(* IEC 61131-3 sources: project_Secure_SCADA/rel_v1.2, 1 file *)

(* ---- rel_v1.2.st ---- *)
FUNCTION_BLOCK TP_WITH_RESET
  VAR_INPUT
    IN : BOOL;
    PT : TIME;
    RESET : BOOL;
  END_VAR
  VAR_OUTPUT
    Q : BOOL;
    ET : TIME := T#0s;
  END_VAR
  VAR
    STATE : SINT := 0;
    PREV_IN : BOOL := FALSE;
    CURRENT_TIME : TIME;
    START_TIME : TIME;
  END_VAR

  (* Pragma to set current time *)
  {__SET_VAR(data__->,CURRENT_TIME,,__CURRENT_TIME)}

  (*Timer block code *)
  IF ((STATE = 0) AND NOT(PREV_IN) AND IN) THEN  (* found rising edge on IN *)
      (* start timer... *)
      STATE := 1;
      Q := TRUE;
      START_TIME := CURRENT_TIME;

  ELSIF (STATE = 1) THEN (* timer counting *)
      IF ((START_TIME + PT) <= CURRENT_TIME) THEN (* timer expired *)
          STATE := 2;
          Q := FALSE;
          ET := PT;
      ELSE (* continue counting *)
          ET := CURRENT_TIME - START_TIME;
      END_IF;
  END_IF;

  IF ((STATE = 2) AND NOT(IN)) THEN
      ET := T#0s;
      STATE := 0;
  END_IF;

  IF (RESET) THEN (* reset pressed *)
    ET := T#0s;
    STATE := 0;
    Q := FALSE;
  END_IF;

  PREV_IN := IN;
END_FUNCTION_BLOCK

PROGRAM aplha
  VAR
    pwr_plant_switch AT %QX0.7 : BOOL;
  END_VAR
  VAR
    pwr_plant : BOOL;
  END_VAR
  VAR
    pwr_gen AT %QX0.0 : BOOL;
    pwr_buildings_on AT %QX0.1 : BOOL;
    pwr_buildings_off AT %QX0.2 : BOOL;
    pwr_hospital_on AT %QX0.3 : BOOL;
    pwr_hospital_off AT %QX0.4 : BOOL;
    alarm AT %QX0.5 : BOOL;
  END_VAR
  VAR
    antenna : BOOL;
    vape_start : BOOL;
    vape_reset : BOOL;
    TP_WITH_RESET0 : TP_WITH_RESET;
    TP0 : TP;
  END_VAR
  VAR
    input_value_gen AT %QW0 : INT := 5000;
    input_value_pwr AT %QW1 : INT := 7000;
    threshold_min_gen AT %QW2 : INT := 2000;
    threshold_min_pwr AT %QW3 : INT := 5000;
  END_VAR
  VAR
    threshold_min_output_gen : BOOL;
    threshold_min_output_pwr : BOOL;
    CTU0 : CTU;
    temp_up : BOOL;
    temp_down : BOOL;
    max_temp : INT := 21;
  END_VAR
  VAR
    current_temp AT %QW4 : INT;
  END_VAR
  VAR
    temp_pulse : BOOL;
    TP2 : TP;
    TP_WITH_RESET1 : TP_WITH_RESET;
    temp_threshold : INT := 6;
  END_VAR
  VAR
    temp_alarm AT %QX0.6 : BOOL;
    max_temp_alarm AT %QX99.7 : BOOL;
  END_VAR
  VAR
    _TMP_GT12_OUT : BOOL;
    _TMP_GT5_OUT : BOOL;
    R_TRIG1 : R_TRIG;
    _TMP_GT22_OUT : BOOL;
  END_VAR

  pwr_plant := threshold_min_output_pwr AND NOT(pwr_plant_switch);
  pwr_gen := threshold_min_output_gen AND NOT(pwr_plant);
  pwr_buildings_on := pwr_plant;
  antenna := pwr_plant;
  pwr_buildings_off := NOT(pwr_plant);
  vape_start := NOT(pwr_plant);
  TP_WITH_RESET0(IN := NOT(vape_reset) AND (pwr_gen OR vape_start), PT := T#2s);
  alarm := TP_WITH_RESET0.Q;
  TP0(IN := TP_WITH_RESET0.Q, PT := T#4s);
  vape_reset := TP0.Q;
  pwr_hospital_on := threshold_min_output_gen AND pwr_gen OR pwr_plant;
  temp_up := NOT(pwr_plant) AND NOT(pwr_gen);
  pwr_hospital_off := NOT(pwr_plant) AND NOT(pwr_gen);
  _TMP_GT12_OUT := GT(input_value_gen, threshold_min_gen);
  threshold_min_output_gen := _TMP_GT12_OUT;
  _TMP_GT5_OUT := GT(input_value_pwr, threshold_min_pwr);
  threshold_min_output_pwr := _TMP_GT5_OUT;
  TP_WITH_RESET1(IN := NOT(temp_pulse) AND temp_up, PT := T#1s);
  TP2(IN := TP_WITH_RESET1.Q, PT := T#2s);
  R_TRIG1(CLK := TP2.Q);
  CTU0(CU := R_TRIG1.Q, R := pwr_hospital_on, PV := max_temp);
  max_temp_alarm := CTU0.Q;
  temp_pulse := TP2.Q;
  current_temp := CTU0.CV;
  _TMP_GT22_OUT := GT(current_temp, temp_threshold);
  temp_alarm := _TMP_GT22_OUT;
END_PROGRAM

CONFIGURATION Config0

  RESOURCE Res0 ON PLC
    TASK task0(INTERVAL := T#20ms,PRIORITY := 0);
    PROGRAM instance0 WITH task0 : aplha;
  END_RESOURCE
END_CONFIGURATION
